FUNCTION_BLOCK ADLINK_IO
  (* Version 1.0, 2005-07-04, Goran Cengic, Chalmers *)
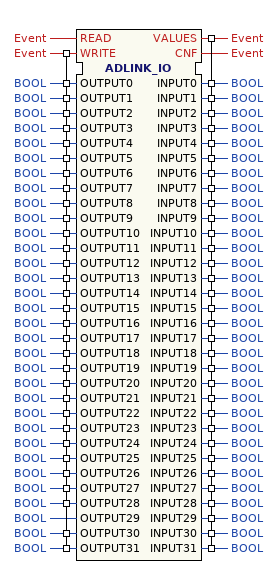
  EVENT_INPUT
    READ;
    WRITE WITH OUTPUT0, OUTPUT1, OUTPUT2, OUTPUT3, OUTPUT4, OUTPUT5, OUTPUT6, OUTPUT7, OUTPUT8, OUTPUT9, OUTPUT10, OUTPUT11, OUTPUT12, OUTPUT13, OUTPUT14, OUTPUT15, OUTPUT16, OUTPUT17, OUTPUT18, OUTPUT19, OUTPUT20, OUTPUT21, OUTPUT22, OUTPUT23, OUTPUT24, OUTPUT25, OUTPUT26, OUTPUT27, OUTPUT28, OUTPUT19, OUTPUT30, OUTPUT31;
  END_EVENT
  EVENT_OUTPUT
    VALUES WITH INPUT0, INPUT1, INPUT2, INPUT3, INPUT4, INPUT5, INPUT6, INPUT7, INPUT8, INPUT9, INPUT10, INPUT11, INPUT12, INPUT13, INPUT14, INPUT15, INPUT16, INPUT17, INPUT18, INPUT19, INPUT20, INPUT21, INPUT22, INPUT23, INPUT24, INPUT25, INPUT26, INPUT27, INPUT28, INPUT29, INPUT30, INPUT31;
    CNF;
  END_EVENT
  VAR_INPUT
    OUTPUT0 : BOOL;
    OUTPUT1 : BOOL;
    OUTPUT2 : BOOL;
    OUTPUT3 : BOOL;
    OUTPUT4 : BOOL;
    OUTPUT5 : BOOL;
    OUTPUT6 : BOOL;
    OUTPUT7 : BOOL;
    OUTPUT8 : BOOL;
    OUTPUT9 : BOOL;
    OUTPUT10 : BOOL;
    OUTPUT11 : BOOL;
    OUTPUT12 : BOOL;
    OUTPUT13 : BOOL;
    OUTPUT14 : BOOL;
    OUTPUT15 : BOOL;
    OUTPUT16 : BOOL;
    OUTPUT17 : BOOL;
    OUTPUT18 : BOOL;
    OUTPUT19 : BOOL;
    OUTPUT20 : BOOL;
    OUTPUT21 : BOOL;
    OUTPUT22 : BOOL;
    OUTPUT23 : BOOL;
    OUTPUT24 : BOOL;
    OUTPUT25 : BOOL;
    OUTPUT26 : BOOL;
    OUTPUT27 : BOOL;
    OUTPUT28 : BOOL;
    OUTPUT29 : BOOL;
    OUTPUT30 : BOOL;
    OUTPUT31 : BOOL;
  END_VAR
  VAR_OUTPUT
    INPUT0 : BOOL;
    INPUT1 : BOOL;
    INPUT2 : BOOL;
    INPUT3 : BOOL;
    INPUT4 : BOOL;
    INPUT5 : BOOL;
    INPUT6 : BOOL;
    INPUT7 : BOOL;
    INPUT8 : BOOL;
    INPUT9 : BOOL;
    INPUT10 : BOOL;
    INPUT11 : BOOL;
    INPUT12 : BOOL;
    INPUT13 : BOOL;
    INPUT14 : BOOL;
    INPUT15 : BOOL;
    INPUT16 : BOOL;
    INPUT17 : BOOL;
    INPUT18 : BOOL;
    INPUT19 : BOOL;
    INPUT20 : BOOL;
    INPUT21 : BOOL;
    INPUT22 : BOOL;
    INPUT23 : BOOL;
    INPUT24 : BOOL;
    INPUT25 : BOOL;
    INPUT26 : BOOL;
    INPUT27 : BOOL;
    INPUT28 : BOOL;
    INPUT29 : BOOL;
    INPUT30 : BOOL;
    INPUT31 : BOOL;
  END_VAR
END_FUNCTION_BLOCK
